Yaskawa INFORM job: FMTV_HOOD_HOLES.JBI

/JOB
//NAME FMTV_HOOD_HOLES
//POS
///NPOS 339,0,0,0,0,0
///TOOL 0
///POSTYPE PULSE
///PULSE
C00000=-63952,-155163,126853,-105316,-81596,-126671
C00001=-74999,-165670,78796,-69370,-117124,-108458
C00002=-100671,-167009,31373,14150,-100380,-66140
C00003=-111612,-167580,-47996,49745,-69453,-48105
C00004=-171050,-113005,-83680,237240,-57967,-79165
C00005=-180792,-99913,-81086,266829,-47651,-77284
C00006=-193514,-80710,-58797,266613,-56361,-78677
C00007=-195482,-77018,-54254,266635,-57690,-78997
C00008=-195481,-77016,-54253,266635,-57688,-78998
C00009=-193514,-80710,-58797,266613,-56361,-78677
C00010=-175084,-106974,-89057,266916,-43709,-76773
C00011=-175084,-106974,-89057,266916,-43709,25582
C00012=-184586,-81176,-43369,303000,-41614,4220
C00013=-187327,-78554,-40483,298175,-44031,5754
C00014=-185640,-80928,-43474,298864,-42902,5541
C00015=-193044,-84392,-49222,294802,-46333,8314
C00016=-194345,-82366,-46638,294398,-47235,8399
C00017=-192583,-85156,-50013,295023,-46048,8222
C00018=-184766,-76589,-46692,296344,-40097,8473
C00019=-186143,-74573,-43862,296019,-41108,8511
C00020=-184808,-76544,-46495,296405,-40154,8424
C00021=-179579,-83617,-56017,298078,-36445,7947
C00022=-175529,-29476,-47093,214499,-119202,11531
C00023=-174045,-31379,-44864,214216,-116880,11352
C00024=-174122,-29277,-42339,214148,-116755,11261
C00025=-174045,-31379,-44864,214216,-116880,11352
C00026=-174857,-30408,-45643,214293,-117938,11351
C00027=-174926,-28222,-42999,214218,-117795,11258
C00028=-174952,-28192,-43040,214223,-117835,11261
C00029=-174857,-30408,-45643,214293,-117938,11351
C00030=-169163,-26488,-47776,216352,-118241,14501
C00031=-169330,-24032,-44705,216236,-118081,14341
C00032=-169409,-24028,-44742,216228,-118130,14320
C00033=-169163,-26488,-47776,216352,-118241,14501
C00034=-168317,-27279,-46764,216223,-117154,14469
C00035=-168493,-24887,-43792,216115,-117011,14314
C00036=-168555,-24918,-43793,216099,-117024,14288
C00037=-168317,-27279,-46764,216223,-117154,14469
C00038=-166675,-46338,-68388,216809,-117337,-83185
C00039=-170592,-31273,-50368,215735,-117864,-85036
C00040=-170845,-27810,-46124,215582,-117678,-85251
C00041=-171153,-26987,-47007,215787,-118517,-85053
C00042=-170940,-26861,-47026,215852,-118493,-84952
C00043=-170771,-26881,-46936,215866,-118380,-84912
C00044=-170341,-27915,-45791,215616,-117298,-85150
C00045=-170341,-27915,-45791,215616,-117298,-85150
C00046=-170598,-28663,-45168,215365,-116822,-85488
C00047=-171710,-28953,-45366,215132,-117222,-85904
C00048=-172120,-28334,-46152,215258,-117975,-85801
C00049=-172046,-28082,-46367,215345,-118142,-85694
C00050=-171153,-26987,-47007,215787,-118517,-85053
C00051=-170845,-27810,-46124,215582,-117678,-85251
C00052=-170335,-34632,-54396,215870,-118002,-84840
C00053=-163472,-58667,-72448,216167,-112526,-59623
C00054=-159889,-60592,-63824,218982,-107558,-59656
C00055=-161475,-59093,-61092,218597,-107773,-60383
C00056=-159889,-60592,-63824,218982,-107558,-59656
C00057=-155484,-51668,-54763,219669,-105650,-58232
C00058=-156903,-50427,-52231,219350,-105782,-58908
C00059=-156924,-50408,-52192,219464,-105818,-58901
C00060=-155484,-51668,-54763,219669,-105650,-58232
C00061=-160193,-50258,-60674,219735,-110615,-58401
C00062=-161277,-49253,-58645,219452,-110702,-58937
C00063=-161532,-49144,-58289,219532,-110761,-59036
C00064=-160193,-50258,-60674,219735,-110615,-58401
C00065=-165027,-58474,-69192,218968,-112777,-59970
C00066=-166595,-56862,-66291,218525,-112960,-60722
C00067=-166619,-56837,-66246,218658,-113009,-60703
C00068=-165027,-58474,-69192,218968,-112777,-59970
C00069=-165775,-68462,-71028,217837,-109745,-61736
C00070=-167158,-67000,-68670,217466,-109985,-62347
C00071=-167158,-67000,-68670,217466,-109985,-62347
C00072=-165775,-68462,-71028,217837,-109745,-61736
C00073=-160304,-70042,-65107,218182,-104382,-61271
C00074=-162126,-68291,-62217,217750,-104720,-62043
C00075=-162156,-68261,-62169,217882,-104780,-62037
C00076=-160304,-70042,-65107,218182,-104382,-61271
C00077=-155047,-61265,-57113,219152,-102508,-59432
C00078=-156899,-59634,-54075,218756,-102774,-60254
C00079=-156927,-59608,-54029,218888,-102824,-60250
C00080=-155047,-61265,-57113,219152,-102508,-59432
C00081=-148945,-65952,-66368,220287,-101543,-56745
C00082=-150681,-42764,-52900,220907,-106323,-55403
C00083=-152138,-41896,-50474,220608,-106389,-56140
C00084=-152138,-41896,-50474,220608,-106389,-56140
C00085=-150511,-43078,-53376,220938,-106305,-55322
C00086=-149673,-36441,-48380,221189,-106617,-54727
C00087=-150870,-35778,-46334,220945,-106638,-55354
C00088=-150870,-35778,-46334,220945,-106638,-55354
C00089=-149512,-36731,-48850,221222,-106611,-54646
C00090=-151375,-39400,-53310,221224,-108118,-54903
C00091=-153272,-38108,-49893,220811,-108175,-55889
C00092=-153272,-38108,-49893,220811,-108175,-55889
C00093=-151375,-39400,-53310,221224,-108118,-54903
C00094=-146437,-42339,-61250,222114,-107730,-52447
C00095=-146437,-42339,-61250,222114,-107730,-52447
C00096=-128609,-128096,-104792,75585,-20102,-123408
C00097=-181435,-102519,-82349,-63516,-17298,-53388
C00098=-194821,-78858,-52778,-63160,-26961,-56004
C00099=-194126,-78083,-50102,-60946,-26989,-57293
C00100=-194191,-78237,-50168,-60922,-27050,-57315
C00101=-194821,-78858,-52778,-63160,-26961,-56004
C00102=-172897,-59551,-49387,-59853,-9599,-56341
C00103=-172115,-58740,-46050,-51884,-9855,-60752
C00104=-172125,-58842,-46111,-51809,-9874,-60794
C00105=-172897,-59551,-49387,-59853,-9599,-56341
C00106=-157127,-85497,-72182,23265,-7402,-101665
C00107=-145667,-81735,-46488,33575,-11186,-97453
C00108=-143333,-80464,-43118,37301,-12939,-99241
C00109=-143333,-80464,-43118,37301,-12939,-99241
C00110=-145667,-81735,-46488,33575,-11186,-97453
C00111=-123031,-69065,-58429,99835,-22269,-133052
C00112=-121442,-67815,-55390,97491,-23251,-131577
C00113=-121442,-67815,-55390,97491,-23251,-131577
C00114=-123031,-69065,-58429,99835,-22269,-133052
C00115=-123031,-69065,-58429,99835,-22269,-133052
C00116=-122934,-59852,-60939,124425,-90658,-109773
C00117=-127441,-38225,-40284,136583,-109952,-109022
C00118=-127460,-34842,-36468,136624,-109816,-108956
C00119=-127444,-37437,-39404,136593,-109923,-109008
C00120=-121374,-42600,-47121,140636,-105859,-101796
C00121=-121545,-40129,-44887,140586,-105896,-101904
C00122=-121374,-42600,-47121,140636,-105859,-101796
C00123=-107803,-42563,-40613,126464,-105757,-97610
C00124=-108355,-39033,-37669,126316,-105639,-97899
C00125=-108355,-39033,-37669,126316,-105639,-97899
C00126=-107803,-42563,-40613,126464,-105757,-97610
C00127=-93834,-42689,-90962,179804,-113224,-85302
C00128=-105765,19381,-33881,179893,-116390,-89971
C00129=-102393,11778,-21533,179924,-106318,-88558
C00130=-101713,7586,-26079,179918,-106449,-88294
C00131=-102393,11778,-21533,179924,-106318,-88558
C00132=-102306,11300,-19332,179937,-104963,-88522
C00133=-101634,7158,-23809,179929,-105084,-88261
C00134=-102306,11300,-19332,179937,-104963,-88522
C00135=-105765,19381,-33881,179893,-116390,-89971
C00136=-93834,-42689,-90962,179804,-113224,-85302
C00137=-59781,-60536,-69399,260621,80630,-31718
C00138=-62508,-52214,-52779,262469,76541,-25832
C00139=-62415,-49824,-49365,262361,76679,-25564
C00140=-62415,-49824,-49365,262361,76679,-25564
C00141=-62504,-52101,-52617,262468,76546,-25817
C00142=-58549,-53537,-51919,262371,79481,-25449
C00143=-58522,-51606,-49202,262304,79556,-25245
C00144=-58522,-51606,-49202,262304,79556,-25245
C00145=-58549,-53537,-51919,262371,79481,-25449
C00146=-64416,-65545,-69188,283326,59987,-31839
C00147=-63305,-63219,-65587,282880,60632,-31356
C00148=-63305,-63219,-65587,282880,60632,-31356
C00149=-64416,-65545,-69188,283326,59987,-31839
C00150=-55532,-76641,-73177,280624,65674,-28972
C00151=-54693,-74520,-70302,280454,66202,-28704
C00152=-54693,-74520,-70302,280454,66202,-28704
C00153=-55532,-76641,-73177,280624,65674,-28972
C00154=-45022,-86307,-75889,279394,72471,-26003
C00155=-44293,-83988,-73115,279367,72951,-25847
C00156=-44293,-83988,-73115,279367,72951,-25847
C00157=-45022,-86307,-75889,279394,72471,-26003
C00158=-32729,-94132,-78053,280192,80576,-23902
C00159=-32141,-91595,-75277,280234,80968,-23818
C00160=-32141,-91595,-75277,280234,80968,-23818
C00161=-32729,-94132,-78053,280192,80576,-23902
C00162=-24425,-111106,-90001,291825,71276,-25961
C00163=-22940,-108544,-87440,291933,72251,-25767
C00164=-22940,-108544,-87440,291933,72251,-25767
C00165=-24425,-111106,-90001,291825,71276,-25961
C00166=-8236,-113831,-89267,287171,87422,-21226
C00167=10775,-104916,-80930,284377,108049,-18729
C00168=10401,-102050,-78115,284278,107813,-18797
C00169=10401,-102050,-78115,284278,107813,-18797
C00170=10775,-104916,-80930,284377,108049,-18729
C00171=29709,-100799,-79130,288814,120388,-17349
C00172=28966,-98094,-76299,288630,119889,-17428
C00173=28966,-98094,-76299,288630,119889,-17428
C00174=29709,-100799,-79130,288814,120388,-17349
C00175=32016,-109007,-86746,289688,121783,-16786
C00176=-36615,-170638,-113836,269613,-10686,-36508
C00177=-42229,-114300,-84368,261462,-117724,-82396
C00178=-38397,-104200,-74915,262649,-115222,-81869
C00179=-37623,-101829,-72496,262838,-114701,-81818
C00180=-37623,-101829,-72496,262838,-114701,-81818
C00181=-38397,-104200,-74915,262649,-115222,-81869
C00182=-18291,-109375,-76711,267330,-102402,-81798
C00183=-17740,-106121,-73615,267480,-102039,-81717
C00184=-17740,-106121,-73615,267480,-102039,-81717
C00185=-18291,-109375,-76711,267330,-102402,-81798
C00186=1406,-118085,-83663,266663,-81028,-81960
C00187=21118,-116630,-84823,264415,-60056,-79456
C00188=19367,-113953,-82276,264068,-61244,-79483
C00189=19367,-113953,-82276,264068,-61244,-79483
C00190=21118,-116630,-84823,264415,-60056,-79456
C00191=30772,-100843,-72407,277185,-68818,-81671
C00192=29937,-97866,-69363,277002,-69385,-81633
C00193=29937,-97866,-69363,277002,-69385,-81633
C00194=30772,-100843,-72407,277185,-68818,-81671
C00195=44618,-93336,-71071,278889,-59419,-80505
C00196=43622,-90694,-68104,278759,-60120,-80529
C00197=43622,-90694,-68104,278759,-60120,-80529
C00198=44618,-93336,-71071,278889,-59419,-80505
C00199=55552,-83923,-68411,279271,-52102,-79076
C00200=54496,-81509,-65390,279284,-52873,-79193
C00201=54496,-81509,-65390,279284,-52873,-79193
C00202=55552,-83923,-68411,279271,-52102,-79076
C00203=64838,-72663,-64629,277066,-44900,-76717
C00204=63791,-70625,-61708,277337,-45678,-76980
C00205=63791,-70625,-61708,277337,-45678,-76980
C00206=64838,-72663,-64629,277066,-44900,-76717
C00207=58121,-61152,-49131,294066,-70164,-79810
C00208=58056,-58581,-45805,294170,-70340,-79987
C00209=58056,-58581,-45805,294170,-70340,-79987
C00210=58121,-61152,-49131,294066,-70164,-79810
C00211=61901,-58869,-48444,295110,-68228,-80109
C00212=61810,-56476,-45321,295216,-68422,-80277
C00213=61810,-56476,-45321,295216,-68422,-80277
C00214=61901,-58869,-48444,295110,-68228,-80109
C00215=63068,-90271,-84517,294574,-66694,-79238
C00216=63068,-90271,-84517,294574,-66694,-79238
C00217=74389,-60227,-82913,260199,-81064,-88249
C00218=88828,16776,-21123,220187,-100034,-97215
C00219=103330,16579,-26620,172321,-117801,-111287
C00220=102267,11737,-15434,173007,-109438,-110969
C00221=101798,8556,-19326,172959,-109710,-111180
C00222=102267,11737,-15434,173007,-109438,-110969
C00223=102364,11880,-12429,172823,-108263,-110867
C00224=101807,8064,-17110,172767,-108591,-111120
C00225=102364,11880,-12429,172823,-108263,-110867
C00226=88828,16776,-21123,220187,-100034,-97215
C00227=74389,-60227,-82913,260199,-81064,-88249
C00228=136659,-58838,-63406,180884,-101749,-96556
C00229=135491,-48710,-56191,180737,-103342,-97020
C00230=135294,-44416,-52670,180712,-103784,-97099
C00231=135491,-48710,-56191,180737,-103342,-97020
C00232=138525,-39763,-45744,180276,-113436,-101343
C00233=138632,-36583,-42428,180305,-113409,-101297
C00234=138525,-39763,-45744,180276,-113436,-101343
C00235=136070,-91121,-88609,179642,-108499,-102328
C00236=146203,-50226,-51119,140750,-105903,55378
C00237=149966,-38550,-50987,139998,-112157,54319
C00238=151678,-37380,-47803,140520,-112179,55250
C00239=151678,-37380,-47803,140520,-112179,55250
C00240=149966,-38550,-50987,139998,-112157,54319
C00241=148114,-35422,-46053,139957,-110649,54063
C00242=149387,-34578,-43662,140328,-110649,54759
C00243=149387,-34578,-43662,140328,-110649,54759
C00244=148114,-35422,-46053,139957,-110649,54063
C00245=149174,-41826,-50787,140329,-110434,54747
C00246=150652,-40808,-48109,140756,-110479,55528
C00247=150652,-40808,-48109,140756,-110479,55528
C00248=149174,-41826,-50787,140329,-110434,54747
C00249=151733,-49626,-56461,141019,-110701,56005
C00250=158636,-59569,-61800,142947,-111851,59155
C00251=160163,-58189,-59142,143442,-112012,59891
C00252=158636,-59569,-61800,142947,-111851,59155
C00253=158669,-49156,-58500,141972,-114778,57796
C00254=159906,-48069,-56166,142405,-114842,58441
C00255=158669,-49156,-58500,141972,-114778,57796
C00256=154267,-50435,-52281,142059,-109876,57748
C00257=155449,-49444,-50143,142421,-109954,58338
C00258=154267,-50435,-52281,142059,-109876,57748
C00259=154038,-59849,-54448,142775,-106817,59020
C00260=155687,-58442,-51689,143253,-107006,59785
C00261=154038,-59849,-54448,142775,-106817,59020
C00262=159168,-68513,-62822,143974,-108812,60786
C00263=160906,-66900,-60015,144514,-109074,61561
C00264=159168,-68513,-62822,143974,-108812,60786
C00265=164034,-67322,-69453,144244,-114029,61030
C00266=165756,-65594,-66495,144841,-114267,61838
C00267=164034,-67322,-69453,144244,-114029,61030
C00268=163326,-57245,-67251,142907,-116988,59293
C00269=165050,-55572,-64048,143546,-117134,60172
C00270=163326,-57245,-67251,142907,-116988,59293
C00271=180397,-114091,-79711,69101,-53018,-107485
C00272=196961,-78271,-44880,75509,-63339,-110306
C00273=197761,-75752,-42055,75692,-63892,-110317
C00274=197761,-75752,-42055,75692,-63892,-110317
C00275=196961,-78271,-44880,75509,-63339,-110306
C00276=185806,-72763,-41746,72640,-55732,-109727
C00277=186722,-70318,-38815,72817,-56390,-109719
C00278=186722,-70318,-38815,72817,-56390,-109719
C00279=185806,-72763,-41746,72640,-55732,-109727
C00280=189635,-71568,-48678,76430,-57144,-112811
C00281=179231,-65491,-42456,73426,-50196,-111506
C00282=180050,-63536,-39986,73503,-50806,-111462
C00283=180050,-63536,-39986,73503,-50806,-111462
C00284=179231,-65491,-42456,73426,-50196,-111506
C00285=182071,-62773,-47735,104117,-67879,-122544
C00286=182888,-60544,-44836,104027,-68363,-122286
C00287=182888,-60544,-44836,104027,-68363,-122286
C00288=182071,-62773,-47735,104117,-67879,-122544
C00289=194490,-71872,-54817,103797,-76592,-126578
C00290=195667,-68002,-49385,103726,-77223,-126066
C00291=195667,-68002,-49385,103726,-77223,-126066
C00292=194490,-71872,-54817,103797,-76592,-126578
C00293=179598,-42258,-42966,113521,-99597,-114012
C00294=179700,-38070,-38198,113562,-99569,-113874
C00295=181154,-37862,-38829,113568,-100686,-113867
C00296=181338,-37937,-38702,113597,-100767,-113786
C00297=181304,-38033,-38513,113620,-100690,-113718
C00298=180012,-38518,-37327,113688,-99517,-113485
C00299=180012,-38518,-37327,113688,-99517,-113485
C00300=179471,-38528,-37194,113664,-99132,-113532
C00301=178777,-38369,-37370,113603,-98745,-113729
C00302=178458,-37839,-38373,113477,-98842,-114180
C00303=179641,-37561,-39180,113450,-99828,-114283
C00304=181206,-37872,-38815,113574,-100715,-113852
C00305=179700,-38070,-38198,113562,-99569,-113874
C00306=179598,-42258,-42966,113521,-99597,-114012
C00307=176925,-65286,-71998,113040,-98908,-14872
C00308=183231,-39863,-38218,113897,-101600,-13174
C00309=183221,-36898,-34820,113931,-101521,-13083
C00310=183231,-39863,-38218,113897,-101600,-13174
C00311=182399,-40302,-36653,114012,-100655,-12790
C00312=182405,-37395,-33332,114042,-100591,-12701
C00313=182399,-40302,-36653,114012,-100655,-12790
C00314=175847,-38325,-40386,113232,-97518,-15289
C00315=175961,-35843,-37510,113255,-97528,-15186
C00316=175847,-38325,-40386,113232,-97518,-15289
C00317=176766,-37742,-41727,113131,-98501,-15649
C00318=176881,-34831,-38335,113161,-98497,-15526
C00319=176766,-37742,-41727,113131,-98501,-15649
C00320=177106,-56055,-48989,79752,-81865,-12300
C00321=181236,-58564,-41667,55788,-33575,-43705
C00322=179783,-57172,-37031,52738,-33702,-41811
C00323=178892,-56256,-34134,50879,-33827,-40665
C00324=178892,-56256,-34134,50879,-33827,-40665
C00325=181236,-58564,-41667,55788,-33575,-43705
C00326=175330,-96871,-115849,113092,-97602,-15922
C00327=185451,-97513,-21096,196210,-113029,-16436
C00328=189111,-94786,-18180,198656,-112401,-15302
C00329=189111,-94786,-18180,198656,-112401,-15302
C00330=185451,-97513,-21096,196210,-113029,-16436
C00331=200506,-101298,-20846,205772,-108297,-12377
C00332=205301,-97221,-16883,208772,-107265,-11031
C00333=200506,-101298,-20846,205772,-108297,-12377
C00334=174969,-92846,-20883,189185,-116469,-19603
C00335=179781,-89231,-16651,192538,-115736,-17995
C00336=174969,-92846,-20883,189185,-116469,-19603
C00337=145149,-108674,-40330,167841,-117405,-30118
C00338=66880,-160385,-79902,187543,-63186,-9823
//INST
///DATE 2022/07/28 12:48
///ATTR SC,RW
///GROUP1 RB1
NOP
MOVJ C00000 VJ=65.00  //HOME
MOVJ C00001 VJ=65.00
MOVJ C00002 VJ=65.00
MOVJ C00003 VJ=65.00  //CENTER
MOVJ C00004 VJ=65.00
MOVL C00005 V=65.0  //ABOVE 30MM
MOVL C00006 V=65.0  //UP TO 30MM
MOVL C00007 V=15.0  //INTO 30MM
FORMCUT FCF#(9)
MOVL C00008 V=65.0
FORMCUT FCF#(9)
MOVL C00009 V=45.0  //OUT OF 30MM
MOVL C00010 V=65.0  //AWAY TO ROTATE
MOVL C00011 V=65.0  //ROTATE
MOVL C00012 V=65.0  //UP TO 1ST 6MM
MOVL C00013 V=15.0  //INTO 1ST 6MM
MOVL C00014 V=45.0  //OUT
MOVL C00015 V=65.0  //UP TO 2ND 6MM
MOVL C00016 V=15.0  //INTO 2ND 6MM
MOVL C00017 V=45.0  //OUT OF 2ND 6MM
MOVL C00018 V=65.0  //UP TO 3RD 6MM
MOVL C00019 V=15.0  //INTO 3RD 6MM
MOVL C00020 V=45.0  //OUT OF 3RD 6MM
MOVL C00021 V=65.0  //AWAY
MOVL C00022 V=65.0
MOVL C00023 V=65.0  //UP TO 1ST 5.75MM
MOVL C00024 V=15.0  //INTO 1ST 5.75MM
MOVL C00025 V=45.0  //OUT OF 1ST 5.75MM
MOVL C00026 V=65.0  //UP TO 2ND 5.75MM
MOVL C00027 V=15.0  //INTO 2ND 5.75MM
MOVL C00028 V=25.0
MOVL C00029 V=45.0  //OUT OF 2ND 5.75MM
MOVL C00030 V=65.0  //UP TO 3RD 5.75MM
MOVL C00031 V=15.0  //INTO 3RD 5.75MM
MOVL C00032 V=25.0
MOVL C00033 V=45.0  //OUT OF 3RD 5.75MM
MOVL C00034 V=65.0  //UP TO 4TH 5.75MM
MOVL C00035 V=15.0  //INTO 4TH 5.75MM
MOVL C00036 V=25.0
MOVL C00037 V=45.0  //OUT OF 4TH 5.75MM
MOVL C00038 V=65.0  //AWAY TO ROTATE
MOVL C00039 V=65.0  //UP TO SHAPE
MOVL C00040 V=15.0  //INTO SHAPE
MOVC C00041 V=15.0  //UP TO EDGE
MOVC C00042 V=15.0
MOVC C00043 V=15.0
MOVL C00044 V=15.0
MOVC C00045 V=15.0
MOVC C00046 V=15.0
MOVC C00047 V=15.0
MOVC C00048 V=15.0
MOVC C00049 V=65.0
MOVL C00050 V=15.0  //END
MOVL C00051 V=65.0  //AWAY FROM EDGE
MOVL C00052 V=65.0  //OUT OF SHAPE
MOVL C00053 V=65.0  //AWAY TO ROTATE
MOVL C00054 V=65.0  //UP TO RIGHT 130MM
MOVL C00055 V=15.0  //INTO RIGHT 130MM
FORMCUT FCF#(11)
MOVL C00056 V=45.0  //OUT OF RIGHT 130MM
MOVL C00057 V=65.0  //UP TO 1ST 7MM
MOVL C00058 V=15.0  //INTO 1ST 7MM
MOVL C00059 V=15.0
MOVL C00060 V=45.0  //OUT OF 1ST 7MM
MOVL C00061 V=65.0  //UP TO 2ND 7MM
MOVL C00062 V=15.0  //INTO 2ND 7MM
MOVL C00063 V=15.0
MOVL C00064 V=45.0  //OUT OF 2ND 7MM
MOVL C00065 V=65.0  //UP TO 3RD 7MM
MOVL C00066 V=15.0  //INTO 3RD 7MM
MOVL C00067 V=15.0
MOVL C00068 V=45.0  //OUT OF 3RD 7MM
MOVL C00069 V=65.0  //UP TO 4TH 7MM
MOVL C00070 V=15.0  //INTO 4TH 7MM
MOVL C00071 V=15.0
MOVL C00072 V=45.0  //OUT OF 4TH 7MM
MOVL C00073 V=65.0  //UP TO 5TH 7MM
MOVL C00074 V=15.0  //INTO 5TH 7MM
MOVL C00075 V=15.0
MOVL C00076 V=45.0  //OUT OF 5TH 7MM
MOVL C00077 V=65.0  //UP TO 6TH 7MM
MOVL C00078 V=15.0  //INTO 6TH 7MM
MOVL C00079 V=15.0
MOVL C00080 V=45.0  //OUT OF 6TH 7MM
MOVL C00081 V=65.0  //AWAY FROM 6TH 7MM
MOVL C00082 V=65.0  //UP TO 1ST 13MM
MOVL C00083 V=15.0  //INTO 1ST 13MM
FORMCUT FCF#(8)
MOVL C00084 V=65.0
FORMCUT FCF#(8)
MOVL C00085 V=45.0  //OUT OF 1ST 13MM
MOVL C00086 V=65.0  //UP TO 2ND 7MM
MOVL C00087 V=15.0  //INTO 2ND 13MM
FORMCUT FCF#(8)
MOVL C00088 V=65.0
FORMCUT FCF#(8)
MOVL C00089 V=45.0  //OUT OF 2ND 13MM
MOVL C00090 V=65.0  //UP TO 40MM
MOVL C00091 V=15.0  //INTO 40MM
FORMCUT FCF#(10)
MOVL C00092 V=65.0
FORMCUT FCF#(10)
MOVL C00093 V=45.0  //OUT OF 40MM
MOVL C00094 V=65.0  //AWAY
MOVJ C00095 VJ=65.00  //AWAY
MOVJ C00096 VJ=65.00  //ROTATE FOR 13MM
MOVL C00097 V=65.0
MOVL C00098 V=65.0  //UP TO 1ST 8MM
MOVL C00099 V=15.0  //INTO 1ST 8MM
MOVL C00100 V=65.0
MOVL C00101 V=45.0  //OUT OF 1ST 8MM
MOVL C00102 V=65.0  //UP TO 2ND 8MM
MOVL C00103 V=15.0  //INTO 2ND 8MM
MOVL C00104 V=15.0
MOVL C00105 V=45.0  //OUT OF 2ND 8MM
MOVL C00106 V=65.0
MOVL C00107 V=65.0  //UP TO 13MM
MOVL C00108 V=15.0  //INTO TO 13MM
FORMCUT FCF#(8)
MOVL C00109 V=65.0
FORMCUT FCF#(8)
MOVL C00110 V=45.0  //OUT OF 1ST 13MM
MOVL C00111 V=65.0  //UP TO 2ND 13MM
MOVL C00112 V=15.0  //INTO 2ND 13MM
FORMCUT FCF#(8)
MOVL C00113 V=65.0
FORMCUT FCF#(8)
MOVL C00114 V=45.0  //OUT OF 2ND 13MM
MOVJ C00115 VJ=65.00
MOVJ C00116 VJ=65.00  //ROTATE TO 7MM
MOVL C00117 V=65.0  //UP TO 1ST 7MM
MOVL C00118 V=15.0  //INTO 1ST 7MM
MOVL C00119 V=45.0  //OUT OF 1ST 7MM
MOVL C00120 V=65.0  //UP TO 2MM
MOVL C00121 V=15.0  //INTO 2ND 7MM
MOVL C00122 V=45.0  //OUT OF 2ND 7MM
MOVL C00123 V=65.0  //UP TO 13MM
MOVL C00124 V=15.0  //INTO 13MM
FORMCUT FCF#(8)
MOVL C00125 V=65.0
FORMCUT FCF#(8)
MOVL C00126 V=65.0  //OUT OF 13MM
MOVL C00127 V=65.0  //SET UP FOR OUTSIDE
MOVL C00128 V=65.0  //TO OUTSIDE
MOVL C00129 V=65.0  //UP TO 1ST 5MM
MOVL C00130 V=15.0  //INTO 1ST 5MM
MOVL C00131 V=45.0  //OUT OF FIRST 5MM
MOVL C00132 V=65.0  //UP TO 2ND 5MM
MOVL C00133 V=15.0  //INTO 2ND 5MM
MOVL C00134 V=45.0  //OUT OF 2ND 5MM
MOVL C00135 V=65.0  //SET UP TO MOVE INSIDE
MOVL C00136 V=65.0  //INSIDE
MOVJ C00137 VJ=65.00  //ROTATE TO RIGHT 11MM
MOVL C00138 V=65.0  //UP TO RIGHT 11MM
MOVL C00139 V=15.0  //RIGHT 11MM
FORMCUT FCF#(7)
MOVL C00140 V=65.0
FORMCUT FCF#(7)
MOVL C00141 V=45.0  //OUT OF RIGHT 11MM
MOVL C00142 V=65.0  //UP TO 2ND 11MM
MOVL C00143 V=15.0  //INTO 2ND 11MM
FORMCUT FCF#(7)
MOVL C00144 V=65.0
FORMCUT FCF#(7)
MOVL C00145 V=45.0  //OUT OF 2ND 11MM
MOVL C00146 V=65.0  //UP TO 3RD 11MM
MOVL C00147 V=15.0  //INTO 3RD 11MM
FORMCUT FCF#(7)
MOVL C00148 V=65.0
FORMCUT FCF#(7)
MOVL C00149 V=45.0  //OUT OF 3RD 11MM
MOVL C00150 V=65.0  //UP TO 4TH 11MM
MOVL C00151 V=15.0  //INTO 4TH 11MM
FORMCUT FCF#(7)
MOVL C00152 V=65.0
FORMCUT FCF#(7)
MOVL C00153 V=45.0  //OUT OF 4TH 11MM
MOVL C00154 V=65.0  //UP TO 5TH 11MM
MOVL C00155 V=15.0  //INTO 5TH 11MM
FORMCUT FCF#(7)
MOVL C00156 V=65.0
FORMCUT FCF#(7)
MOVL C00157 V=45.0  //OUT OF 5TH 11MM
MOVL C00158 V=65.0  //UP TO 6TH 11MM
MOVL C00159 V=15.0  //INTO 6TH 11MM
FORMCUT FCF#(7)
MOVL C00160 V=65.0
FORMCUT FCF#(7)
MOVL C00161 V=45.0  //OUT OF 6TH 11MM
MOVL C00162 V=65.0  //UP TO 7TH 11MM
MOVL C00163 V=15.0  //INTO 7TH 11MM
FORMCUT FCF#(7)
MOVL C00164 V=65.0
FORMCUT FCF#(7)
MOVL C00165 V=45.0  //OUT OF 7TH 11MM
MOVL C00166 V=65.0  //OVER CORNER
MOVL C00167 V=65.0  //UP TO 8TH 11MM
MOVL C00168 V=45.0  //INTO 8TH 11MM
FORMCUT FCF#(7)
MOVL C00169 V=65.0
FORMCUT FCF#(7)
MOVL C00170 V=45.0  //OUT OF 8TH 11MM
MOVL C00171 V=65.0  //UP TO 9TH 11MM
MOVL C00172 V=15.0  //INTO 9TH 11MM
FORMCUT FCF#(7)
MOVL C00173 V=65.0
FORMCUT FCF#(7)
MOVL C00174 V=45.0  //OUT OF 9TH 11MM
MOVJ C00175 VJ=65.00  //ABOVE 9TH
MOVJ C00176 VJ=65.00  //ROTATE B AXIS
MOVJ C00177 VJ=65.00  //ABOVE 10TH
MOVJ C00178 VJ=65.00  //UP TO 11TH
MOVL C00179 V=15.0  //INTO 10TH 11MM
FORMCUT FCF#(7)
MOVL C00180 V=65.0
FORMCUT FCF#(7)
MOVL C00181 V=45.0  //OUT OF 10TH 11MM
MOVL C00182 V=65.0  //UP TO 11TH 11MM
MOVL C00183 V=15.0  //INTO 11TH 11MM
FORMCUT FCF#(7)
MOVL C00184 V=65.0
FORMCUT FCF#(7)
MOVL C00185 V=45.0  //OUT OF 11TH 11MM
MOVL C00186 V=65.0  //ABOVE CORNER
MOVL C00187 V=65.0  //UP TO 12TH 11MM
MOVL C00188 V=15.0  //INTO 12TH 11MM
FORMCUT FCF#(7)
MOVL C00189 V=65.0
FORMCUT FCF#(7)
MOVL C00190 V=45.0  //OUT OF 12TH 11MM
MOVL C00191 V=65.0  //UP TO 13TH 11MM
MOVL C00192 V=15.0  //INTO 13TH 11MM
FORMCUT FCF#(7)
MOVL C00193 V=65.0
FORMCUT FCF#(7)
MOVL C00194 V=45.0  //OUT OF 13TH 11MM
MOVL C00195 V=65.0  //UP TO 14TH 11MM
MOVL C00196 V=15.0  //INTO 14TH 11MM
FORMCUT FCF#(7)
MOVL C00197 V=65.0
FORMCUT FCF#(7)
MOVL C00198 V=45.0  //OUT OF 14TH 11MM
MOVL C00199 V=65.0  //UP TO 15TH 11MM
MOVL C00200 V=15.0  //INTO 15TH 11MM
FORMCUT FCF#(7)
MOVL C00201 V=65.0
FORMCUT FCF#(7)
MOVL C00202 V=45.0  //OUT OF 15TH 11MM
MOVL C00203 V=65.0  //UP TO 16TH 11MM
MOVL C00204 V=15.0  //INTO 16TH 11MM
FORMCUT FCF#(7)
MOVL C00205 V=65.0
FORMCUT FCF#(7)
MOVL C00206 V=45.0  //OUT OF 16TH 11MM
MOVL C00207 V=65.0  //UP TO 17TH 11MM
MOVL C00208 V=15.0  //INTO 17TH 11MM
FORMCUT FCF#(7)
MOVL C00209 V=65.0
FORMCUT FCF#(7)
MOVL C00210 V=45.0  //OUT OF 17TH 11MM
MOVL C00211 V=65.0  //UP TO 18TH 11MM
MOVL C00212 V=15.0  //INTO 18TH 11MM
FORMCUT FCF#(7)
MOVL C00213 V=65.0
FORMCUT FCF#(7)
MOVL C00214 V=45.0  //OUT OF 18TH 11MM
MOVL C00215 V=65.0  //AWAY FROM PART
MOVJ C00216 VJ=65.00
MOVJ C00217 VJ=65.00  //ROTATE TO MOVE OUTSIDE
MOVJ C00218 VJ=65.00  //OUTSIDE OF PART
MOVJ C00219 VJ=65.00  //ABOVE LEFT 5MM
MOVL C00220 V=65.0  //UP TO TOP LEFT 5MM
MOVL C00221 V=15.0  //INTO TOP LEFT 5MM
MOVL C00222 V=45.0  //OUT OF TOP LEFT 5MM
MOVL C00223 V=65.0  //UP TO BOTTOM LEFT 5MM
MOVL C00224 V=15.0  //INTO BOTTOM LEFT 5MM
MOVL C00225 V=45.0  //OUT OF BOTTOM LEFT 5MM
MOVJ C00226 VJ=65.00  //ROTATE TO GET INSIDE
MOVJ C00227 VJ=65.00  //INSIDE PART
MOVJ C00228 VJ=65.00  //ROTATE TO LEFT 7MM
MOVL C00229 V=65.0  //UP TO FRONT LEFT 7MM
MOVL C00230 V=15.0  //INTO FRONT LEFT 7MM
MOVL C00231 V=45.0  //OUT OF FRONT LEFT 7MM
MOVL C00232 V=65.0  //UP TO BACK LEFT 7MM
MOVL C00233 V=15.0  //INTO BACK LEFT 7MM
MOVL C00234 V=45.0  //OUT OF BACK LEFT 7MM
MOVL C00235 V=65.0  //AWAY FROM 7MM
MOVL C00236 V=65.0  //ROTATE SQUARE TO LEFT HEADLIGHT
MOVL C00237 V=65.0  //UP TO LEFT 40MM
MOVL C00238 V=15.0  //INTO LEFT 40MM
FORMCUT FCF#(10)
MOVL C00239 V=65.0
FORMCUT FCF#(10)
MOVL C00240 V=45.0  //OUT OF LEFT 40MM
MOVL C00241 V=65.0  //UP TO 1ST LEFT 13MM
MOVL C00242 V=15.0  //INTO 1ST LEFT 13MM
FORMCUT FCF#(8)
MOVL C00243 V=65.0
FORMCUT FCF#(8)
MOVL C00244 V=45.0  //OUT OF 1ST LEFT 13MM
MOVL C00245 V=65.0  //UP TO 2ND LEFT 13MM
MOVL C00246 V=15.0  //INTO 2ND LEFT 13MM
FORMCUT FCF#(8)
MOVL C00247 V=65.0
FORMCUT FCF#(8)
MOVL C00248 V=45.0  //OUT OF 2ND LEFT 13MM
MOVL C00249 V=65.0  //OVER CORNER
MOVL C00250 V=65.0  //UP TO LEFT 130MM
MOVL C00251 V=15.0  //INTO LEFT 130MM
FORMCUT FCF#(11)
MOVL C00252 V=45.0  //OUT OF LEFT 130MM
MOVL C00253 V=65.0  //UP TO 1ST 7MM
MOVL C00254 V=15.0  //INTO 1ST 7MM
MOVL C00255 V=45.0  //OUT OF
MOVL C00256 V=65.0  //UP TO
MOVL C00257 V=15.0  //INTO 2ND 7MM
MOVL C00258 V=45.0  //OUT OF
MOVL C00259 V=65.0  //UP TO
MOVL C00260 V=15.0  //INTO 3RD 7MM
MOVL C00261 V=45.0  //OUT OF
MOVL C00262 V=65.0  //UP TO
MOVL C00263 V=15.0  //INTO 4TH 7MM
MOVL C00264 V=45.0  //OUT OF
MOVL C00265 V=65.0  //UP TO
MOVL C00266 V=15.0  //INTO 5TH 7MM
MOVL C00267 V=45.0  //OUT OF
MOVL C00268 V=65.0  //UP TO
MOVL C00269 V=15.0  //INTO 6TH 7MM
MOVL C00270 V=45.0  //OUT OF
MOVJ C00271 VJ=65.00  //ROTATE TO 10MM
MOVL C00272 V=65.0  //UP TO 1ST 10MM
MOVL C00273 V=15.0  //INTO 1ST 10MM
FORMCUT FCF#(6)
MOVL C00274 V=65.0
FORMCUT FCF#(6)
MOVL C00275 V=45.0  //OUT OF 1ST 10MM
MOVL C00276 V=65.0  //UP TO 2ND 10MM
MOVL C00277 V=15.0  //INTO 2ND 10MM
FORMCUT FCF#(6)
MOVL C00278 V=65.0
FORMCUT FCF#(6)
MOVL C00279 V=45.0  //OUT OF 2ND 10MM
MOVL C00280 V=65.0  //AWAY
MOVL C00281 V=65.0  //UP TO 3RD 10MM
MOVL C00282 V=15.0  //INTO 3RD 10MM
FORMCUT FCF#(6)
MOVL C00283 V=65.0
FORMCUT FCF#(6)
MOVL C00284 V=45.0  //OUT OF 3RD 10MM
MOVL C00285 V=65.0  //UP TO 4TH
MOVL C00286 V=15.0  //INTO 4TH 1OMM
FORMCUT FCF#(6)
MOVL C00287 V=65.0
FORMCUT FCF#(6)
MOVL C00288 V=45.0  //OUT OF 4TH
MOVL C00289 V=65.0  //UP TO 5TH
MOVL C00290 V=15.0  //INTO 5TH
FORMCUT FCF#(6)
MOVL C00291 V=65.0
FORMCUT FCF#(6)
MOVL C00292 V=45.0  //OUT OF 5TH
MOVL C00293 V=65.0  //UP TO SHAPE
MOVL C00294 V=15.0  //INTO SHAPE
MOVC C00295 V=15.0
MOVC C00296 V=15.0
MOVC C00297 V=15.0
MOVL C00298 V=15.0
MOVC C00299 V=15.0
MOVC C00300 V=15.0
MOVC C00301 V=15.0
MOVC C00302 V=15.0
MOVC C00303 V=15.0
MOVL C00304 V=15.0
MOVL C00305 V=15.0  //CENTER OF SHAPE
MOVL C00306 V=65.0  //OUT OF SHAPE
MOVL C00307 V=65.0  //AWAY TO ROTATE
MOVL C00308 V=65.0  //UP TO 1ST 5.75MM
MOVL C00309 V=15.0  //INTO 1ST 5.75MM
MOVL C00310 V=45.0  //OUT OF 1ST 5.75
MOVL C00311 V=65.0  //UP TO 2ND 5.75MM
MOVL C00312 V=15.0  //INTO 2ND 5.75MM
MOVL C00313 V=45.0  //OUT OF 2ND 5.75MM
MOVL C00314 V=65.0  //UP TO 5.75MM
MOVL C00315 V=15.0  //INTO 3RD 5.75
MOVL C00316 V=45.0  //OUT OF 3RD 5.75MM
MOVL C00317 V=65.0  //UP TO 4TH 5.75MM
MOVL C00318 V=15.0  //INTO 4TH 5.75MM
MOVL C00319 V=45.0  //OUT OF 4TH 5.75
MOVL C00320 V=65.0
MOVL C00321 V=65.0
MOVL C00322 V=65.0
MOVL C00323 V=15.0  //INTO 8MM
FORMCUT FCF#(5)
MOVL C00324 V=65.0
FORMCUT FCF#(5)
MOVL C00325 V=45.0
MOVL C00326 V=65.0  //AWAY FROM PART
MOVL C00327 V=65.0  //UP TO 11MM
MOVL C00328 V=15.0  //INTO 11MM
FORMCUT FCF#(7)
MOVL C00329 V=65.0
FORMCUT FCF#(7)
MOVL C00330 V=45.0  //OUT OF 11MM
MOVL C00331 V=65.0  //UP TO 1ST 5.5MM
MOVL C00332 V=15.0  //INTO 1ST 5.5MM
MOVL C00333 V=45.0  //OUT OF 1ST 5.5MM
MOVL C00334 V=65.0  //UP TO 2ND 5.5MM
MOVL C00335 V=15.0  //INTO 2ND 5.5MM
MOVL C00336 V=45.0  //OUT OF 2ND 5.5MM
MOVL C00337 V=65.0  //AWAY
MOVJ C00338 VJ=65.00
END
